TYPE TYP_RGB_LED_CHANNEL :
STRUCT
	Out : TYP_RGB_LED_CHANNEL_OUT;
END_STRUCT
END_TYPE

(* stored: Version 1.1.0.1, ProductVersion 3.1.4024.12
   DUT TYP_RGB_LED_CHANNEL: Id {bffec77c-1362-4faf-a753-b6bb2056ffb7} *)
